			(*MetaDaten sammeln*)
			IF bStoreMetaDataInFile THEN
				FOR iMetaID :=0 TO 499 BY 1 DO
					IF arrMetaID[iMetaID]=arrDP_ID_buffer[iBuffer] THEN
						iMetaID:=500;
					ELSIF arrMetaID[iMetaID]='' THEN
						arrMetaID[iMetaID]:=arrDP_ID_buffer[iBuffer] ;
						arrMetaData[iMeta]:=arrLogDatapoints[iBuffer];
						IF arrMetaData[iMeta].sID='' THEN
							arrMetaData[iMeta].sID:=arrMetaData[iMeta].sDescription;
						END_IF
						IF arrMetaData[iMeta].sUnit='' THEN
							arrMetaData[iMeta].sUnit:='-';
						END_IF
						iMeta:=iMeta+1;
						iMetaID:=500;
			//			bStoreMeta:=TRUE;
					END_IF
				END_FOR
			END_IF
			IF iBuffer <499 THEN
				IF arrLogDatapoints[iBuffer+1].sDescription ='' AND arrLogDatapoints[iBuffer+1].sID = '' THEN
					iBuffer:=500;
				END_IF		
			END_IF				
		ELSE
			iBuffer:=500;
		END_IF
	END_FOR
ELSE
	bArrayStored:=FALSE;
END_IF

(*MetaDatenBuffern*)
IF arrMetaData[0].sDescription<>'' AND arrMetaDataBuffer[0].sDescription='' THEN
	arrMetaDataBuffer:=arrMetaData;
	iMeta:=0;
	arrMetaData:=arrMetaDataEmpty;	
END_IF

(*MetaDaten in Datei speichern*)
IF arrMetaDataBuffer[0].sDescription<>'' AND sFolderPath <>'' THEN
	CASE iState_StoreMeta OF
		0:	// Datei anlegen
			(*fbFormatMetaFilepath(
				sFormat	:= '%S\%S_%S',
				arg1	:= F_STRING(sFolderPath),
				arg2	:= F_STRING(sLMeasurement_date),
				arg3	:= F_STRING(sMetaFileName),
				sOut	=> sFilePathMeta,
				bError	=> bFormatMetaFilepath_error,
				nErrId	=> nFormatMetaFilepath_errID
			);*)
			sFilePathMeta:=CONCAT(sFolderPath,'\');
			sFilePathMeta:=CONCAT(sFilePathMeta,sLMeasurement_date);
			sFilePathMeta:=CONCAT(sFilePathMeta,sMetaFileName);
			//sFilePathMeta:=CONCAT(sFilePathMeta,'_MetaData.txt');
			fbFileOpenMeta(
				bExecute:=FALSE,
				);
			
			fbFileOpenMeta(
				sNetID:='',
				sPathName:=sFilePathMeta,
				nMode:=FOPEN_MODEAPPEND,
				//ePath:=ePath,
				bExecute:=TRUE,
				tTimeout:=T#5S,
				);
			iState_StoreMeta:=iState_StoreMeta+1;
			
		1:	// warten bis Funktionsbaustein fertig
			fbFileOpenMeta(
				bExecute:=FALSE,
				);
			IF NOT fbFileOpenMeta.bBusy THEN
				IF fbFileOpenMeta.bError THEN
					iFileOpenMeta_errID:=fbFileOpenMeta.nErrId;
					iState_StoreMeta:=0;
				ELSE
					hFileMeta:=fbFileOpenMeta.hFile;
					iFileOpenMeta_errID:=fbFileOpenMeta.nErrId;
					iState_StoreMeta:=10;
				END_IF	
			END_IF
			
		10:	// String vorbereiten
			IF arrMetaDataBuffer[iMetaBuffer].sDescription <> ''  THEN
				CASE iMetaInfo OF
					0:  sStringMeta:=CONCAT('ID=',arrMetaDataBuffer[iMetaBuffer].sID);
						sStringMeta:=CONCAT(sStringMeta,'$0A');
					1:	sStringMeta:=CONCAT('Description=',arrMetaDataBuffer[iMetaBuffer].sDescription);
						sStringMeta:=CONCAT(sStringMeta,'$0A');
					2:	sStringMeta:=CONCAT('Unit=',arrMetaDataBuffer[iMetaBuffer].sUnit);	
						sStringMeta:=CONCAT(sStringMeta,'$0A$0A');		
				END_CASE
				IF iMetaInfo>=2 THEN
					iMetaInfo:=0;
					iMetaBuffer:=iMetaBuffer+1;
				ELSE
					iMetaInfo:=iMetaInfo+1;
				END_IF	
				iState_StoreMeta:=11;
			ELSE
				iState_StoreMeta:=20;
			END_IF			
		
		11:	// Tabelle schreiben
		fbFilePutsMeta(
			sNetID:='',
			hfile:=hFileMeta,
			sLine:=sStringMeta,
			bExecute:=TRUE,
			bBusy=>bPutsMeta_busy,
			bError=>bPutsMeta_error,
			nErrId=>iPutsMeta_errorID
			);
			
		// wenn Funktionsbaustein fertig, zum nächsten Datenpunkt springen			
		IF NOT bPutsMeta_busy OR bPutsMeta_error THEN
			fbFilePutsMeta(
				bExecute:=FALSE,
				bBusy=>bPutsMeta_busy,
				bError=>bPutsMeta_error,
				nErrId=>iPutsMeta_errorID
				);
				
			IF bPutsMeta_error THEN
				nErrorMeta_LogError:=nErrorMEta_LogError+1;
			END_IF
				
			MEMSET(ADR(sStringMeta),0,255);
			iState_StoreMeta:=10;
		END_IF			
			
			
		20: // Datei schließen
			fbFileCloseMeta(
				bExecute:=FALSE,
				);
			fbFileCloseMeta(
				sNetId:='',
				hFile:=hFileMeta,
				bExecute:=TRUE,
				tTimeout:=,
				);
			iState_StoreMeta:=iState_StoreMeta+1;
			
		21: // warten bis Baustein fertig ist
			fbFileCloseMeta(
				bExecute:=FALSE,
				);
			IF NOT fbFileCloseMeta.bBusy THEN		
				IF fbFileCloseMeta.bError THEN
					iFileCloseMeta_errID:=fbFileCloseMeta.nErrId;
				END_IF
					iFileCloseMeta_errID:=fbFileCloseMeta.nErrId;
					iState_StoreMeta:=30;
			END_IF
			
		30: // Speichervorgang abgschlossen
			//bSafe_Table:=FALSE;
			iMetaBuffer:=0;
			arrMetaDataBuffer:=arrMetaDataEmpty;
			iState_StoreMeta:=0;
	END_CASE
END_IF

// Messwerte abspeichern, sofern nicht gerade die Meassdatendatei getauscht wird
IF bLogging AND hFile<>0 THEN
	bLogging_activ:=TRUE;
	CASE iStateLogging OF
	0:	// Datenpunktstring bauen
		// Dezimalunkt durch Komma ersetzen im Messwert
		IF FIND(arrDP_Value_buffer[iDatapoint_Log],'.') <>0 THEN
			arrDP_Value_buffer[iDatapoint_Log]:=REPLACE(arrDP_Value_buffer[iDatapoint_Log],',',1,FIND(arrDP_Value_buffer[iDatapoint_Log],'.')); 
		END_IF
		
		// String zusammensetzen 
			IF bLogUtcTime THEN
				// UTC
				fbFormatMeasString(
					sFormat	:= '%S%S%S%S',
					arg1	:= F_STRING(sMeasurement_date),
					arg2	:= F_STRING(sSpaces),
					arg3	:= F_STRING(sMeasurement_time),
					arg4	:= F_STRING(sDelimiter),
					sOut	=> sMeasString_temp,
					bError	=> bFormatMeasString_error,
					nErrId	=> nFormatMeasString_errID
					);
					
				IF bFormatTimestamp_error THEN
					nError_Logging:=nError_Logging+1;
				END_IF
			END_IF
			
			IF bLogLocalTime THEN
				// lokale Zeit
				fbFormatMeasString(
					sFormat	:= '%S%S%S%S%S',
					arg1	:= F_STRING(sMeasString_temp),
					arg2	:= F_STRING(sLMeasurement_date),
					arg3	:= F_STRING(sSpaces),
					arg4	:= F_STRING(sLMeasurement_time),
					arg5	:= F_STRING(sDelimiter),
					sOut	=> sMeasString_temp,
					bError	=> bFormatMeasString_error,
					nErrId	=> nFormatMeasString_errID
					);
				
				IF bFormatTimestamp_error THEN
					nError_Logging:=nError_Logging+1;
				END_IF	
			END_IF
				
			// Datenpunkte
			fbFormatMeasString(
				sFormat	:= '%S%S%S%S',
				arg1	:= F_STRING(sMeasString_temp),
				arg2	:= F_STRING(arrDP_ID_buffer[iDatapoint_Log]),
				arg3	:= F_STRING(sDelimiter),
				arg4	:= F_STRING(arrDP_Value_buffer[iDatapoint_Log]),
				sOut	=> sMeasString_temp,
				bError	=> bFormatMeasString_error,
				nErrId	=> nFormatMeasString_errID
				);

			IF bFormatTimestamp_error THEN
				nError_Logging:=nError_Logging+1;
			END_IF		
				
		// String für CSV vorbereiten
		fb_CSVbuffer(
			eCmd:=eCmd,
			putValue:=sMeasString_temp,
			pValue:=0,
			cbValue:=0,
			bCRLF:=bCRLF,
			pBuffer:=ADR(sMeasString),
			cbBuffer:=SIZEOF(sMeasString),
			cbSize=>iSize_buffer
			);
		
		sMeasString_temp:='';	
			
		// Zeilenende hinzufügen
		MEMSET(ADR(sMeasString)+iSize_buffer-2,9,1);
		sMeasString:=REPLACE(sMeasString,'$0A',2,FIND(sMeasString,'$09$0A'));
		iStateLogging:=1;
		
	1:	//Datenpunktstring schreiben
		fbFilePuts(
			sNetID:='',
			hfile:=hFile,
			sLine:=sMeasString,
			bExecute:=TRUE,
			bBusy=>bPuts_busy,
			bError=>bPuts_error,
			nErrId=>iPuts_errorID
			);
			
		bWatchdogDPwrite:=FALSE;
			
		// wenn Funktionsbaustein fertig, zum nächsten Datenpunkt springen			
		IF NOT bPuts_busy OR bPuts_error THEN
			fbFilePuts(
				bExecute:=FALSE,
				bBusy=>bPuts_busy,
				bError=>bPuts_error,
				nErrId=>iPuts_errorID
				);
				
			IF bPuts_error THEN
				nError_Logging:=nError_Logging+1;
			END_IF
				
			iDatapoint_Log:=iDatapoint_Log+1;
			MEMSET(ADR(sMeasString),0,255);
			IF arrDP_ID_buffer[iDatapoint_Log]<>'' AND iDatapoint_Log<>500 THEN
				iStateLogging:=0;
			ELSE // falls dies der letzte Datenpunkt war, Speicherzyklus beenden
				IF arrDP_ID_buffer[0]='' THEN
					iNumberOfLoggedDP:= 0;
				ELSE
					iNumberOfLoggedDP:= iDatapoint_Log;				
				END_IF
				arrDP_ID_buffer:=arrTMAXempty;
				arrDP_Value_buffer:=arrTMAXempty;
				iDatapoint_Log:=0;
				iStateLogging:=0;
				bLogging:=FALSE;
				bLogging_activ:=FALSE;
			END_IF
		END_IF
	END_CASE
END_IF

IF tLogCycleTime<T#100MS THEN
	tWatchdogDPwrite_Time:=T#500MS;
ELSE
	tWatchdogDPwrite_Time:=2*tLogCycleTime;
END_IF

fbWatchdogDPwrite(IN:=bWatchdogDPwrite, PT:= tWatchdogDPwrite_Time, Q=> , ET=> );
IF fbWatchdogDPwrite.Q THEN
	bWatchdogDPwrite:=FALSE;
	nError_Logging:=nError_Logging+1;
ELSE
	bWatchdogDPwrite:=TRUE;
END_IF

END_FUNCTION_BLOCK

// Datenlogger/FB/FB_TIME
FUNCTION_BLOCK FB_TIME
VAR
	// Allgemein
	iStateZeit					:INT;
	
	// Zeitzonenermittlung
	iState_Timezone				:INT;
	FB_GetTimeZone				:FB_GetTimeZoneInformation;
	bGetTimeZone_busy			:BOOL;
	bGetTimeZone_error			:BOOL;
	nGetTimeZone_errID			:UDINT;
	tzGetTimeZone_Info  		:ST_TimeZoneInformation;
	tzGetTimeZone_InfoTc  		:ST_TimeZoneInformation;
	nTimeZonebias				:DINT;
	
	// Erkennung der Zeitzonenänderung
	FB_TimezoneChange_Timeout	:TON;
	nTimeZoneChanging_Timeout	:UINT;
	nTimeout					:TIME:=T#1S;

	// Zeitermittlung Windows Zeit
	fbGetTime					:NT_GetTime;
	bGetTime_busy				:BOOL;
	bGetTime_error				:BOOL;
	nGetTime_errID				:UDINT;
	nGetTime_errCounter			:UDINT;
	fbTimeToUTC					:FB_TzSpecificLocalTimeToSystemTime;	
	
	// Zeitermittlung TwinCat Zeit	
	fbGetSystemTime				:GetSystemTime;
	tfTcDate					:T_Filetime;
	tTcDate						:TIMESTRUCT;
	fbUTCtoLTime				:FB_SystemTimeToTzSpecificLocalTime;
	bTimeZoneInitialized		:BOOL;
END_VAR

VAR_IN_OUT 
// ehemals Globale Variablen
	// Time	
	bUseTcTime					:BOOL;									(*Zeitbasis: fortlaufende TwinCAT-Uhr initialisiert durch Windows*)
	// Time local
	tLDate						:TIMESTRUCT;							(*aktuelles Datum lokal*)
	tfLDate						:T_Filetime;							(*aktuelles Datum lokal*)
	sLYear						:T_MaxString;							(*aktuelles Jahr lokal als String*)
	sLMonth						:T_MaxString;							(*aktueller Monat lokal als String*)
	sLDay						:T_MaxString;							(*aktueller Tag lokal als String*)
	sLHour						:T_MaxString;							(*aktuelle Stunde lokal als String*)
	sLMinute					:T_MaxString;							(*aktuelle Minute lokal als String*)
	sLSecond					:T_MaxString;							(*aktuelle Sekunde lokal als String*)
	sLMilliSecond				:T_MaxString;							(*aktulle Millisekunde lokal als String*)
	
	// Time UTC
	tDate						:TIMESTRUCT;							(*aktuelles Datum UTC*)
	tfDate						:T_Filetime;							(*aktuelles Datum UTC*)
	wDate						:LWORD;									(*aktuelles Datum UTC*)
	sYear						:T_MaxString;							(*aktuelles Jahr UTC als String*)
	sMonth						:T_MaxString;							(*aktueller Monat UTC als String*)
	sDay						:T_MaxString;							(*aktueller Tag UTC als String*)
	sHour						:T_MaxString;							(*aktuelle Stunde UTC als String*)
	sMinute						:T_MaxString;							(*aktuelle Minute UTC als String*)
	sSecond						:T_MaxString;							(*aktuelle Sekunde UTC als String*)
	sMilliSecond				:T_MaxString;							(*aktulle Millisekunde UTC als String*)
	
	// Errohandling
	nError_Time					:UINT;
END_VAR

IF NOT bUseTcTime THEN // USE Windows-Zeitbasis
	// Ermittlung der Zeitzoneninformation
		CASE iState_Timezone OF
		0:	
			FB_GetTimeZone(
				sNetID:= , 
				bExecute:=TRUE , 
				tTimeout:=T#3S , 
				bBusy=> bGetTimeZone_busy, 
				bError=> bGetTimeZone_error, 
				nErrID=> nGetTimeZone_errID, 
				tzID=> , 
				tzInfo=> );
		
			iState_Timezone:=1;
			
		1:		
			FB_GetTimeZone(
				sNetID:= , 
				bExecute:=FALSE , 
				tTimeout:=T#3S , 
				bBusy=> bGetTimeZone_busy, 
				bError=> bGetTimeZone_error, 
				nErrID=> nGetTimeZone_errID, 
				tzID=> , 
				tzInfo=> //tzGetTimeZone_Info
				);
				
			IF (bGetTimeZone_busy=FALSE) THEN
				IF NOT bGetTimeZone_error AND FB_GetTimeZone.tzInfo.standardName<>'' THEN
					tzGetTimeZone_Info:=FB_GetTimeZone.tzInfo;
					iState_Timezone:=0;
					IF tzGetTimeZone_Info.bias<>nTimeZonebias THEN
						nTimeZonebias:=tzGetTimeZone_Info.bias;
						iStateZeit:=3;
					END_IF
				ELSE
					nError_Time:=nError_Time+1;
					iState_Timezone:=0;
				END_IF
			END_IF
		END_CASE
	
	
		CASE iStateZeit OF
		0:
			(*Zeit auslesen*)
			fbGetTime(
				NETID		:= '',
				START		:= TRUE,
				TMOUT		:= T#2s,
				BUSY		=>bGetTime_busy ,
				ERR			=>bGetTime_error ,
				ERRID		=>nGetTime_errID ,
				TIMESTR		=>
			);
			
			fbGetTime(
				START		:= FALSE,
			);
			fbGetTime(
				START		:= TRUE,
			);
			iStateZeit:=1;
			
		1:
			fbGetTime(
				START		:= FALSE,
				BUSY		=>bGetTime_busy ,
				ERR			=>bGetTime_error ,
				ERRID		=>nGetTime_errID ,
			);
			
			IF NOT fbGetTime.BUSY AND NOT fbGetTime.ERR  THEN
				(*aktuelles Datum lokal*)
				tLDate	:= fbGetTime.TIMESTR;
				tfLDate	:= SYSTEMTIME_TO_FILETIME(tLDATE);
				
				(* lokale Zeit in String übersetzen*)
				sLYear			:= DWORD_TO_DECSTR(tLDate.wYear, 4);
				sLMonth			:= DWORD_TO_DECSTR(tLDate.wMonth, 2);
				sLDay			:= DWORD_TO_DECSTR(tLDate.wDay, 2);
				sLHour			:= DWORD_TO_DECSTR(tLDate.wHour, 2);
				sLMinute		:= DWORD_TO_DECSTR(tLDate.wMinute, 2);
				sLSecond		:= DWORD_TO_DECSTR(tLDate.wSecond, 2);
				sLMilliSecond	:= DWORD_TO_DECSTR(tLDate.wMilliseconds, 3);
				
				(*aktuelles Datum UTC*)
				fbTimeToUTC(
					in:= tlDate, 
					tzInfo:= tzGetTimeZone_Info, 
					out=> tDate, 
					eTzID=> , 
					bB=> );
				tfDate	:=	SYSTEMTIME_TO_FILETIME(tDate);
				MEMCPY(ADR(wDate)+4,ADR(tfDate.dwHighDateTime),4);
				MEMCPY(ADR(wDate),ADR(tfDate.dwLowDateTime),4);		
				
				(*UTC Zeit in String übersetzen*)
				sYear			:= DWORD_TO_DECSTR(tDate.wYear, 4);
				sMonth			:= DWORD_TO_DECSTR(tDate.wMonth, 2);
				sDay			:= DWORD_TO_DECSTR(tDate.wDay, 2);
				sHour			:= DWORD_TO_DECSTR(tDate.wHour, 2);
				sMinute			:= DWORD_TO_DECSTR(tDate.wMinute, 2);
				sSecond			:= DWORD_TO_DECSTR(tDate.wSecond, 2);
				sMilliSecond	:= DWORD_TO_DECSTR(tDate.wMilliseconds, 3);
				
				iStateZeit:=0;	
			ELSIF NOT fbGetTime.BUSY AND fbGetTime.ERR  THEN
				iStateZeit:=0;
				nError_Time:=nError_Time+1;
				nGetTime_errCounter:=nGetTime_errCounter+1;		
			END_IF
		
		3:	// Timeout bei Zeitzonenänderung
			FB_TimezoneChange_Timeout(IN:= TRUE, PT:= nTimeout , Q=> , ET=> );
			IF FB_TimezoneChange_Timeout.Q THEN
				iStateZeit:=0;
				FB_TimezoneChange_Timeout(IN:= FALSE, PT:= nTimeout , Q=> , ET=> );
				fbGetTime(
					START		:= FALSE,
				);	
			END_IF
		END_CASE		
ELSE	// USE TwinCat Zeitbasis
	CASE iState_Timezone OF
	// Ermittlung der Zeitzoneninformation
	0:	
		FB_GetTimeZone(
			sNetID:= , 
			bExecute:=TRUE , 
			tTimeout:=T#3S , 
			bBusy=> bGetTimeZone_busy, 
			bError=> bGetTimeZone_error, 
			nErrID=> nGetTimeZone_errID, 
			tzID=> , 
			tzInfo=> );
	
		iState_Timezone:=1;
		
	1:		
		FB_GetTimeZone(
			sNetID:= , 
			bExecute:=FALSE , 
			tTimeout:=T#3S , 
			bBusy=> bGetTimeZone_busy, 
			bError=> bGetTimeZone_error, 
			nErrID=> nGetTimeZone_errID, 
			tzID=> , 
			tzInfo=> tzGetTimeZone_Info
			);
			
		IF (bGetTimeZone_busy=FALSE) THEN
			IF NOT bGetTimeZone_error THEN
				tzGetTimeZone_InfoTc:=FB_GetTimeZone.tzInfo;
				iState_Timezone:=0;
			ELSE
				nError_Time:=nError_Time+1;
				iState_Timezone:=0;
			END_IF
			bTimeZoneInitialized :=TRUE;
		END_IF	
	END_CASE	
	
	IF bTimeZoneInitialized THEN
	// Errechnung der UTC auf Basis der TwinCat Zeit
		(*aktuelles Datum UTC TwinCat*)
		fbGetSystemTime(timeLoDW=>tfTcDate.dwLowDateTime , timeHiDW=> tfTcDate.dwHighDateTime);
		tTcDate	:=	FILETIME_TO_SYSTEMTIME(tfTcDate);
		
		(*aktuelles Datum lokal*)
		fbUTCtoLTime(
			in:= tTcDate, 
			tzInfo:= tzGetTimeZone_InfoTc, 
			out=> tLDate, 
			eTzID=> , 
			bB=> );		
		tfLDate	:= SYSTEMTIME_TO_FILETIME(tLDATE);
		
		(* lokale Zeit in String übersetzen*)
		sLYear			:= DWORD_TO_DECSTR(tLDate.wYear, 4);
		sLMonth			:= DWORD_TO_DECSTR(tLDate.wMonth, 2);
		sLDay			:= DWORD_TO_DECSTR(tLDate.wDay, 2);
		sLHour			:= DWORD_TO_DECSTR(tLDate.wHour, 2);
		sLMinute		:= DWORD_TO_DECSTR(tLDate.wMinute, 2);
		sLSecond		:= DWORD_TO_DECSTR(tLDate.wSecond, 2);
		sLMilliSecond	:= DWORD_TO_DECSTR(tLDate.wMilliseconds, 3);
		
		(*aktuelles Datum UTC*)	
		tfDate:=tfTcDate;	
		tDate	:=	FILETIME_TO_SYSTEMTIME(tfDate);
		MEMCPY(ADR(wDate)+4,ADR(tfDate.dwHighDateTime),4);
		MEMCPY(ADR(wDate),ADR(tfDate.dwLowDateTime),4);		
		
		(*UTC Zeit in String übersetzen*)
		sYear			:= DWORD_TO_DECSTR(tDate.wYear, 4);
		sMonth			:= DWORD_TO_DECSTR(tDate.wMonth, 2);
		sDay			:= DWORD_TO_DECSTR(tDate.wDay, 2);
		sHour			:= DWORD_TO_DECSTR(tDate.wHour, 2);
		sMinute			:= DWORD_TO_DECSTR(tDate.wMinute, 2);
		sSecond			:= DWORD_TO_DECSTR(tDate.wSecond, 2);
		sMilliSecond	:= DWORD_TO_DECSTR(tDate.wMilliseconds, 3);
	END_IF	
END_IF

END_FUNCTION_BLOCK

// Datenlogger/FB_Datenlogger
FUNCTION_BLOCK FB_Datenlogger
VAR_INPUT
	arrLogDatapoints			:ARRAY [0..499] OF Log_Datapoint;		(*Logging Input*)
//	arrDatenpunkt_ID			:ARRAY [0..99] OF T_MaxString;			(*Beschreibung der Datenpunkte*)
//	arrDatenpunkt				:ARRAY [0..99] OF T_MaxString;			(*Messwerte der Datenpunkte*)
	sPathName				 	:T_MaxString:='C:\Messdaten\'; 			(*Pfad der Messdaten festlegen (default: C:\Messdaten\, nur der letzte Unterordner wird (falls nicht vorhanden) erstellt*)
	tZykluszeit					:TIME:=T#10S;							(*Messzykluszeit (default: 10s), 0 entspricht so schnell wie möglich*)
	bExecute					:BOOL:=TRUE;							(*externe (De)aktivierung der Loggingfunktion (default: aktiviert)*)
	bUseTwinCatTimeBase			:BOOL:=FALSE;							(*Zeit auf Basis der fortlaufenden TwinCAT-Uhr intialisiert durch Windows (default: deaktiviert); zu verwenden wenn die WindowsZeit nicht netzwerkseitig synchronisiert wird*)
	bLocalTimeLogging			:BOOL:=TRUE;							(*lokale Zeit mitloggen (default: aktiviert)*)
	bOldOutputFile				:BOOL:=FALSE;							(*FALSE(default)OutputFile:"idTABvalue"; TRUE(oldFormat):OutputFile: "DescriptionTAB[unit]TABvalue --> no Meta"*)
END_VAR
VAR_OUTPUT
	bArrayStored				:BOOL;									(*Flag, Loggarray in Puffer übertragen*)
	sLogFilePath				:STRING;								(*Path of actual LogFile*)
	arrLoggedDatapoints			:ARRAY [0..499] OF Log_Datapoint;		(*Array of Logged Datapoints*)
	iNumberOfLoggedDatapoints	:INT;									(*information of Loged Datapoints*)
	nErrorCounter				:UINT;									(*Anzahl aufgelaufener Fehler*)
END_VAR
VAR
	FB_TIME						:FB_TIME;								(*Funktionsbaustein für die Zeitsteuerung*)
	FB_FOLDER					:FB_FOLDER;								(*Funktionsbaustein für die Ordnererstellung*)
	FB_FILE						:FB_FILE;								(*Funktionsbaustein für die Dateierstellung*)
	FB_LOGGING					:FB_LOGGING;							(*Funktionsbaustein für das Schreiben der Messdaten*)
END_VAR
VAR
	bUtcTimeLogging				:BOOL:=TRUE;							(*UTC mitloggen (default: aktiviert)*)
// ehemals Globale Variablen
// General	
	arrDatapoint_ID				:ARRAY [0..499] OF T_MaxString;			(*Beschreibung der Datenpunkte*)
	arrDatapoint_Value			:ARRAY [0..499] OF T_MaxString;			(*Messwerte der Datenpunkte*)
	sDataPath					:T_MaxString:='C:\Messdaten\'; 			(*Pfad der Messdaten*)
	tLogCycleTime				:TIME:=T#10S;							(*Messzyklusvorgabe*)

// Time	
	bUseTcTime					:BOOL;									(*Zeitbasis: fortlaufende TwinCAT-Uhr initialisiert durch Windows*)
	// Time local
	tLDate						:TIMESTRUCT;							(*aktuelles Datum lokal*)
	tfLDate						:T_Filetime;							(*aktuelles Datum lokal*)
	sLYear						:T_MaxString;							(*aktuelles Jahr lokal als String*)
	sLMonth						:T_MaxString;							(*aktueller Monat lokal als String*)
	sLDay						:T_MaxString;							(*aktueller Tag lokal als String*)
	sLHour						:T_MaxString;							(*aktuelle Stunde lokal als String*)
	sLMinute					:T_MaxString;							(*aktuelle Minute lokal als String*)
	sLSecond					:T_MaxString;							(*aktuelle Sekunde lokal als String*)
	sLMilliSecond				:T_MaxString;							(*aktulle Millisekunde lokal als String*)
	
	// Time UTC
	tDate						:TIMESTRUCT;							(*aktuelles Datum UTC*)
	tfDate						:T_Filetime;							(*aktuelles Datum UTC*)
	wDate						:LWORD;									(*aktuelles Datum UTC*)
	sYear						:T_MaxString;							(*aktuelles Jahr UTC als String*)
	sMonth						:T_MaxString;							(*aktueller Monat UTC als String*)
	sDay						:T_MaxString;							(*aktueller Tag UTC als String*)
	sHour						:T_MaxString;							(*aktuelle Stunde UTC als String*)
	sMinute						:T_MaxString;							(*aktuelle Minute UTC als String*)
	sSecond						:T_MaxString;							(*aktuelle Sekunde UTC als String*)
	sMilliSecond				:T_MaxString;							(*aktulle Millisekunde UTC als String*)
	
	
// File and Folder
	// allgemein
	iStateFolder				:INT;									(*Case Auswahl der Ordnererzeugung*)
	arrLastFolder				:ARRAY [0..2] OF STRING;				(*letzter erzeugter Datumsordner*)
	sFolderPath					:T_MaxString;							(*Pfad, zum Messdatenordner*)
	sFilePath					:T_MaxString;							(*Pfad zur Messdatendatei*)
	
	// Statusvariablen der Dateierstellung
	sLastFile_Changed			:T_MaxString:='99';						(*Minute der letzten Änderung des verwedndeten Datenfiles*)
	sLastFile_Opened			:T_MaxString:='99';						(*Minute des letzten geöffneten Datenfiles*)

	// Dateireferenzen	
	hFile						:UINT;									(*Referenz der aktuellen Messdatendatei*)
	hFile_Close					:UINT;									(*Referenz der zu schließenden Messdatendatei*)
	arrhFile_Open				:ARRAY [0..10] OF UINT;					(*Referenz-Array der geöffneten Messdatendatein*)		

// Logging
	wNextMeasurement			:LWORD;									(*Zeit des nächsten vorgesehenen Loggings*)
	bLogging_activ				:BOOL;									(*Flag; zeigt an, ob gerade Werte geschrieben werden*)
	bLogUtcTime					:BOOL;									(*UTC Zeit mitloggen*)
	bLogLocalTime				:BOOL;									(*lokale Zeit mitloggen*)
	
// Errohandling
	nError_Time					:UINT;
	nError_Folder				:UINT;
	nError_File_Open			:UINT;
	nError_File_Close			:UINT;	
	nError_File_Change			:UINT;		
	nError_Logging				:UINT;	
	nError_Datalogger			:UINT;
END_VAR

// Verknüpfung der Eingänge auf die globalen Variablen
// zur Nutzung des Funktionsbausteins aus in bestehenden Projekten
//arrDatapoint_ID			:=arrDatenpunkt_ID;
//arrDatapoint_Value		:=arrDatenpunkt;
sDataPath				:=sPathName;
tLogCycleTime			:=tZykluszeit;
bLogUtcTime				:=bUtcTimeLogging;			
bLogLocalTime			:=bLocalTimeLogging;
bUseTcTime				:=bUseTwinCatTimeBase;		

FB_TIME(
	bUseTcTime:= bUseTcTime, 
	tLDate:= tLDate, 
	tfLDate:= tfLDate, 
	sLYear:= sLYear, 
	sLMonth:= sLMonth, 
	sLDay:= sLDay, 
	sLHour:= sLHour, 
	sLMinute:= sLMinute, 
	sLSecond:= sLSecond, 
	sLMilliSecond:= sLMilliSecond, 
	tDate:= tDate, 
	tfDate:= tfDate, 
	wDate:= wDate, 
	sYear:= sYear, 
	sMonth:= sMonth, 
	sDay:= sDay, 
	sHour:= sHour, 
	sMinute:= sMinute, 
	sSecond:= sSecond, 
	sMilliSecond:= sMilliSecond, 
	nError_Time:= nError_Time);
	
IF NOT bExecute  THEN // Rücksetzen des Loggers in Ausgangsstellung
	IF bLogging_activ THEN
		FB_LOGGING(
			arrLogDatapoints:=arrLogDatapoints,
			bArrayStored:=bArrayStored,
//			arrDatapoint_ID:= arrDatapoint_ID, 
//			arrDatapoint_Value:= arrDatapoint_Value, 
			tLogCycleTime:= tLogCycleTime, 
			sLYear:= sLYear, 
			sLMonth:= sLMonth, 
			sLDay:= sLDay, 
			sLHour:= sLHour, 
			sLMinute:= sLMinute, 
			sLSecond:= sLSecond, 
			sLMilliSecond:= sLMilliSecond, 
			wDate:= wDate, 
			sYear:= sYear, 
			sMonth:= sMonth, 
			sDay:= sDay, 
			sHour:= sHour, 
			sMinute:= sMinute, 
			sSecond:= sSecond, 
			sMilliSecond:= sMilliSecond, 
			sFolderPath:=sFolderPath,
			hFile:= hFile, 
			wNextMeasurement:= wNextMeasurement, 
			bLogging_activ:= bLogging_activ, 
			bLogUtcTime:= bLogUtcTime, 
			bLogLocalTime:= bLogLocalTime,
			bOldOutputFile :=bOldOutputFile,
			nError_Logging:= nError_Logging, 
			nError_Datalogger:= nError_Datalogger,
			iNumberOfLoggedDP=>iNumberOfLoggedDatapoints,
			arrLoggedDatapoints=>arrLoggedDatapoints);
			
	ELSIF hFile <> 0 THEN
		// Datei freigeben	
		sLastFile_Changed			:='97';
		sLastFile_Opened			:='97';
		hFile_Close					:=hFile;
		FB_FILE(
			tfDate:= tfDate, 
			sYear:= sYear, 
			sMonth:= sMonth, 
			sDay:= sDay, 
			sHour:= sHour, 
			sMinute:= sMinute, 
			sSecond:= sSecond, 
			sMilliSecond:= sMilliSecond, 
			sFolderPath:= sFolderPath, 
			sFilePath:= sFilePath, 
			sLastFile_Changed:= sLastFile_Changed, 
			sLastFile_Opened:= sLastFile_Opened, 
			hFile:= hFile, 
			hFile_Close:= hFile_Close, 
			arrhFile_Open:= arrhFile_Open, 
			bLogging_activ:= bLogging_activ, 
			nError_File_Open:= nError_File_Open, 
			nError_File_Close:= nError_File_Close, 
			nError_File_Change:= nError_File_Change);
		
		// Werte für Loggerneustart Rücksetzen
		wNextMeasurement			:=0;
		iStateFolder				:=0;
		arrLastFolder[0]			:='0';
		arrLastFolder[1]			:='0';
		arrLastFolder[2]			:='0';
		sFolderPath					:='';
		sFilePath					:='';
		bArrayStored:=TRUE;
	ELSE
		bArrayStored:=FALSE;	
	END_IF

ELSE	// Aufruf der Funktionsbausteine
	FB_FOLDER(
		sDataPath:= sDataPath, 
		tfDate:= tfDate, 
		wDate:= wDate, 
		sYear:= sYear, 
		iStateFolder:= iStateFolder, 
		arrLastFolder:= arrLastFolder, 
		sFolderPath:= sFolderPath, 
		nError_Folder:= nError_Folder);
	FB_FILE(
		tfDate:= tfDate, 
		sYear:= sYear, 
		sMonth:= sMonth, 
		sDay:= sDay, 
		sHour:= sHour, 
		sMinute:= sMinute, 
		sSecond:= sSecond, 
		sMilliSecond:= sMilliSecond, 
		sFolderPath:= sFolderPath, 
		sFilePath:= sFilePath, 
		sLastFile_Changed:= sLastFile_Changed, 
		sLastFile_Opened:= sLastFile_Opened, 
		hFile:= hFile, 
		hFile_Close:= hFile_Close, 
		arrhFile_Open:= arrhFile_Open, 
		bLogging_activ:= bLogging_activ, 
		nError_File_Open:= nError_File_Open, 
		nError_File_Close:= nError_File_Close, 
		nError_File_Change:= nError_File_Change);
		
	FB_LOGGING(
		arrLogDatapoints:=arrLogDatapoints,
		bArrayStored:=bArrayStored,
//		arrDatapoint_ID:= arrDatapoint_ID, 
//		arrDatapoint_Value:= arrDatapoint_Value, 
		tLogCycleTime:= tLogCycleTime, 
		sLYear:= sLYear, 
		sLMonth:= sLMonth, 
		sLDay:= sLDay, 
		sLHour:= sLHour, 
		sLMinute:= sLMinute, 
		sLSecond:= sLSecond, 
		sLMilliSecond:= sLMilliSecond, 
		wDate:= wDate, 
		sYear:= sYear, 
		sMonth:= sMonth, 
		sDay:= sDay, 
		sHour:= sHour, 
		sMinute:= sMinute, 
		sSecond:= sSecond, 
		sMilliSecond:= sMilliSecond, 
		sFolderPath:=sFolderPath,
		hFile:= hFile, 
		wNextMeasurement:= wNextMeasurement, 
		bLogging_activ:= bLogging_activ, 
		bLogUtcTime:= bLogUtcTime, 
		bLogLocalTime:= bLogLocalTime, 
		bOldOutputFile:=bOldOutputFile,
		nError_Logging:= nError_Logging, 
		nError_Datalogger:= nError_Datalogger,
		iNumberOfLoggedDP=>iNumberOfLoggedDatapoints,
		arrLoggedDatapoints=>arrLoggedDatapoints);		
END_IF

IF sFilePath <> '' THEN
	sLogFilePath:=sFilePath;
END_IF
nError_Datalogger:=nError_Time+nError_Folder+nError_File_Open+nError_File_Change+nError_File_Close+nError_Logging;
nErrorCounter	:=nError_Datalogger;

END_FUNCTION_BLOCK

// Functions/FUN_ByteArrToString
FUNCTION FUN_ByteArrToString :STRING
VAR_INPUT
	arrTempBytes:ARRAY [0..7] OF BYTE;
	iDatatyp 	:Datatyp;
	bHex		:BOOL;
END_VAR
VAR
	sTempBYTE :BYTE;
	sTempWORD :WORD;
	sTempDWORD :DWORD;
	sTempSINT :SINT;
	sTempINT :INT;
	sTempDINT :DINT;
	sTempLINT :LINT;
	sTempUSINT :USINT;
	sTempUINT :UINT;
	sTempUDINT :UDINT;
	sTempULINT :ULINT;
	sTempREAL :REAL;
	sTempLREAL :LREAL;
	sTempBOOL :BYTE;
	sTempEnum :BYTE;
END_VAR

CASE iDatatyp OF
0: // NO_DATA_TYP_DEFINED

1:	// BYTE
	MEMCPY(ADR(sTempBYTE),ADR(arrTempBytes),SIZEOF(sTempBYTE));
	IF bHex THEN
		FUN_ByteArrToString := BYTE_TO_HEXSTR(sTempBYTE,0,FALSE);
	ELSE
		FUN_ByteArrToString := BYTE_TO_STRING(sTempBYTE);
	END_IF
		
	
2: // WORD
	MEMCPY(ADR(sTempWORD), ADR(arrTempBytes), SIZEOF(sTempWORD));	
	IF bHex THEN
		FUN_ByteArrToString := WORD_TO_HEXSTR(sTempWORD,0,FALSE);
	ELSE
		FUN_ByteArrToSTring := WORD_TO_STRING(sTempWORD);
	END_IF
	
3: // DWORD
	MEMCPY(ADR(sTempDWORD), ADR(arrTempBytes), SIZEOF(sTempDWORD));	
	IF bHex THEN
		FUN_ByteArrToString := DWORD_TO_HEXSTR(sTempDWORD,0,FALSE);
	ELSE
		FUN_ByteArrToSTring := DWORD_TO_STRING(sTempDWORD);
	END_IF

4: // SINT
	MEMCPY(ADR(sTempSINT), ADR(arrTempBytes), SIZEOF(sTempSINT));	
	IF bHex THEN
		FUN_ByteArrToSTring := DATA_TO_HEXSTR(pData := ADR(sTempSINT), cbData:=SIZEOF(sTempSINT),bLoCase:=FALSE);
	ELSE
		FUN_ByteArrToSTring := SINT_TO_STRING(sTempSINT);		
	END_IF
		
5: // INT
	MEMCPY(ADR(sTempINT), ADR(arrTempBytes), SIZEOF(sTempINT));	
	IF bHex THEN
		FUN_ByteArrToSTring := DATA_TO_HEXSTR(pData := ADR(sTempINT), cbData:=SIZEOF(sTempINT),bLoCase:=FALSE);
	ELSE
		FUN_ByteArrToSTring := INT_TO_STRING(sTempINT);		
	END_IF
	
6: // DINT
	MEMCPY(ADR(sTempDINT), ADR(arrTempBytes), SIZEOF(sTempDINT));	
	IF bHex THEN
		FUN_ByteArrToSTring := DATA_TO_HEXSTR(pData := ADR(sTempDINT), cbData:=SIZEOF(sTempDINT),bLoCase:=FALSE);
	ELSE
		FUN_ByteArrToSTring := DINT_TO_STRING(sTempDINT);		
	END_IF
	
7: // LINT
	MEMCPY(ADR(sTempLINT), ADR(arrTempBytes), SIZEOF(sTempLINT));	
	IF bHex THEN
		FUN_ByteArrToSTring := DATA_TO_HEXSTR(pData := ADR(sTempLINT), cbData:=SIZEOF(sTempLINT),bLoCase:=FALSE);
	ELSE
		FUN_ByteArrToSTring := LINT_TO_STRING(sTempLINT);
	END_IF
	
8: // USINT
	MEMCPY(ADR(sTempUSINT), ADR(arrTempBytes), SIZEOF(sTempUSINT));	
	IF bHex THEN
		FUN_ByteArrToSTring := DATA_TO_HEXSTR(pData := ADR(sTempUSINT), cbData:=SIZEOF(sTempUSINT),bLoCase:=FALSE);
	ELSE
		FUN_ByteArrToSTring := USINT_TO_STRING(sTempUSINT);		
	END_IF
	
9: // UINT
	MEMCPY(ADR(sTempUINT), ADR(arrTempBytes), SIZEOF(sTempUINT));	
	IF bHex THEN
		FUN_ByteArrToSTring := DATA_TO_HEXSTR(pData := ADR(sTempUINT), cbData:=SIZEOF(sTempUINT),bLoCase:=FALSE);
	ELSE
		FUN_ByteArrToSTring := UINT_TO_STRING(sTempUINT);		
	END_IF
	
10: // UDINT
	MEMCPY(ADR(sTempUDINT), ADR(arrTempBytes), SIZEOF(sTempUDINT));	
	IF bHex THEN
		FUN_ByteArrToSTring := DATA_TO_HEXSTR(pData := ADR(sTempUDINT), cbData:=SIZEOF(sTempUDINT),bLoCase:=FALSE);
	ELSE
		FUN_ByteArrToSTring := UDINT_TO_STRING(sTempUDINT);
	END_IF
	
11: // ULINT
	MEMCPY(ADR(sTempULINT), ADR(arrTempBytes), SIZEOF(sTempULINT));	
	IF bHex THEN
		FUN_ByteArrToSTring := DATA_TO_HEXSTR(pData := ADR(sTempULINT), cbData:=SIZEOF(sTempULINT),bLoCase:=FALSE);
	ELSE
		FUN_ByteArrToSTring := ULINT_TO_STRING(sTempULINT);		
	END_IF
	
12: // REAL
	MEMCPY(ADR(sTempREAL), ADR(arrTempBytes), SIZEOF(sTempREAL));	
	IF bHex THEN
		FUN_ByteArrToSTring := DATA_TO_HEXSTR(pData := ADR(sTempREAL), cbData:=SIZEOF(sTempREAL),bLoCase:=FALSE);
	ELSE
		FUN_ByteArrToSTring := REAL_TO_STRING(sTempREAL);		
	END_IF
	
13: // LREAL
	MEMCPY(ADR(sTempLREAL), ADR(arrTempBytes), SIZEOF(sTempLREAL));	
	IF bHex THEN
		FUN_ByteArrToSTring := DATA_TO_HEXSTR(pData := ADR(sTempLREAL), cbData:=SIZEOF(sTempLREAL),bLoCase:=FALSE);
	ELSE
		FUN_ByteArrToSTring := LREAL_TO_STRING(sTempLREAL);		
	END_IF
	
14: // BOOL->Byte
	MEMCPY(ADR(sTempBOOL), ADR(arrTempBytes), SIZEOF(sTempBOOL));	
	IF bHex THEN
		FUN_ByteArrToSTring := DATA_TO_HEXSTR(pData := ADR(sTempBOOL), cbData:=SIZEOF(sTempBOOL),bLoCase:=FALSE);
	ELSE
		FUN_ByteArrToSTring := BYTE_TO_STRING(sTempBOOL);		
	END_IF
	
15: // ENUM->Byte
	MEMCPY(ADR(sTempENUM), ADR(arrTempBytes), SIZEOF(sTempENUM));	
	IF bHex THEN
		FUN_ByteArrToSTring := DATA_TO_HEXSTR(pData := ADR(sTempENUM), cbData:=SIZEOF(sTempENUM),bLoCase:=FALSE);
	ELSE
		FUN_ByteArrToSTring := BYTE_TO_STRING(sTempENUM);	
	END_IF
	
END_CASE

END_FUNCTION

// Functions/FUN_DatatypSize
FUNCTION FUN_DatatypSize : UINT
VAR_INPUT
	iDatatyp :Datatyp;
END_VAR
VAR
END_VAR

CASE iDatatyp OF
0: // NOT DEFINED
	FUN_DatatypSize:=0;	
1: // BYTE
	FUN_DatatypSize:=1;
2: // WORD
	FUN_DatatypSize:=2;
3: // DWORD
	FUN_DatatypSize:=4;
4: // SINT
	FUN_DatatypSize:=1;
5: // INT
	FUN_DatatypSize:=2;
6: // DINT
	FUN_DatatypSize:=4;
7: // LINT
	FUN_DatatypSize:=8;
8: // USINT
	FUN_DatatypSize:=1;
9: // UINT
	FUN_DatatypSize:=2;
10: // UDINT
	FUN_DatatypSize:=4;
11: // ULINT
	FUN_DatatypSize:=8;
12: // REAL
	FUN_DatatypSize:=4;
13: // LREAL
	FUN_DatatypSize:=8;
14: // BOOL->Byte
	FUN_DatatypSize:=1;
15: // ENUM->Byte
	FUN_DatatypSize:=1;
END_CASE

END_FUNCTION

// Functions/FUN_StringToByteArr
FUNCTION FUN_StringToByteArr : ARRAY [0..7] OF BYTE
VAR_INPUT
	sTempValue	:STRING;
	iDatatyp 	:Datatyp;
END_VAR
VAR
	sTempBYTE :BYTE;
	sTempWORD :WORD;
	sTempDWORD :DWORD;
	sTempSINT :SINT;
	sTempINT :INT;
	sTempDINT :DINT;
	sTempLINT :LINT;
	sTempUSINT :USINT;
	sTempUINT :UINT;
	sTempUDINT :UDINT;
	sTempULINT :ULINT;
	sTempREAL :REAL;
	sTempLREAL :LREAL;
	sTempBOOL :BYTE;
	sTempEnum :BYTE;
END_VAR

CASE iDatatyp OF
0: // NO_DATA_TYP_DEFINED

1:	// BYTE
	sTempBYTE := STRING_TO_BYTE(sTempValue);
	MEMCPY(ADR(FUN_StringToByteArr),ADR(sTempBYTE),SIZEOF(sTempBYTE));
2: // WORD
	sTempWORD := STRING_TO_WORD(sTempValue);
	MEMCPY(ADR(FUN_StringToByteArr),ADR(sTempWORD),SIZEOF(sTempWORD));
3: // DWORD
	sTempDWORD := STRING_TO_DWORD(sTempValue);
	MEMCPY(ADR(FUN_StringToByteArr),ADR(sTempDWORD),SIZEOF(sTempDWORD));
4: // SINT
	sTempSINT := STRING_TO_SINT(sTempValue);
	MEMCPY(ADR(FUN_StringToByteArr),ADR(sTempSINT),SIZEOF(sTempSINT));
5: // INT
	sTempINT := STRING_TO_INT(sTempValue);
	MEMCPY(ADR(FUN_StringToByteArr),ADR(sTempINT),SIZEOF(sTempINT));
6: // DINT
	sTempDINT := STRING_TO_DINT(sTempValue);
	MEMCPY(ADR(FUN_StringToByteArr),ADR(sTempDINT),SIZEOF(sTempDINT));
7: // LINT
	sTempLINT := STRING_TO_LINT(sTempValue);
	MEMCPY(ADR(FUN_StringToByteArr),ADR(sTempLINT),SIZEOF(sTempLINT));
8: // USINT
	sTempUSINT := STRING_TO_USINT(sTempValue);
	MEMCPY(ADR(FUN_StringToByteArr),ADR(sTempUSINT),SIZEOF(sTempUSINT));
9: // UINT
	sTempUINT := STRING_TO_UINT(sTempValue);
	MEMCPY(ADR(FUN_StringToByteArr),ADR(sTempUINT),SIZEOF(sTempUINT));
10: // UDINT
	sTempUDINT := STRING_TO_UDINT(sTempValue);
	MEMCPY(ADR(FUN_StringToByteArr),ADR(sTempUDINT),SIZEOF(sTempUDINT));
11: // ULINT
	sTempULINT := STRING_TO_ULINT(sTempValue);
	MEMCPY(ADR(FUN_StringToByteArr),ADR(sTempULINT),SIZEOF(sTempULINT));
12: // REAL
	sTempREAL := STRING_TO_REAL(sTempValue);
	MEMCPY(ADR(FUN_StringToByteArr),ADR(sTempREAL),SIZEOF(sTempREAL));
13: // LREAL
	sTempLREAL := STRING_TO_LREAL(sTempValue);
	MEMCPY(ADR(FUN_StringToByteArr),ADR(sTempLREAL),SIZEOF(sTempLREAL));
14: // BOOL->Byte
	sTempBOOL := STRING_TO_BYTE(sTempValue);
	MEMCPY(ADR(FUN_StringToByteArr),ADR(sTempBOOL),SIZEOF(sTempBOOL));
15: // ENUM->Byte
	sTempEnum := STRING_TO_BYTE(sTempValue);
	MEMCPY(ADR(FUN_StringToByteArr),ADR(sTempEnum),SIZEOF(sTempEnum));	
END_CASE

END_FUNCTION

// Timetable/FB_TimeTable
FUNCTION_BLOCK FB_TimeTable
VAR_INPUT
//	nInputValue					:LREAL;		
	arrTimeControl				:ARRAY [0..49] OF Struct_TimeTable;
END_VAR

VAR_OUTPUT
	nOutputValue				:LREAL;
	bValueChanged				:BOOL;
END_VAR
VAR
	wLastMinute					:WORD;
	iRow						:INT;
	
	// Zeitermittlung Windows Zeit
	iStateZeit					:INT;
	fbGetTime					:NT_GetTime;
	bGetTime_busy				:BOOL;
	bGetTime_error				:BOOL;
	nGetTime_errID				:UDINT;
	
	// Time local
	tLDate						:TIMESTRUCT;				(*aktuelles Datum lokal*)
	

	// Tabelle abspeichern
	arrTimeControlSafed			:ARRAY [0..49] OF Struct_TimeTable;
	bSafe_Table					:BOOL;
	iState_safe					:INT;
	sFilePath					:T_MaxString:='C:\Timetable.txt';
	// Datei öffnen
	bOpenFile					:BOOL;
	fbFileOpen					:FB_FileOpen;
	iFileOpen_errID				:UDINT;
	hFile						:UINT;
	// Datei schließen
	bCloseFile					:BOOL;
	fbFileClose					:FB_FileClose;
	iFileClose_errID			:UDINT;
	// Daten schreiben
	iRow_safe					:INT;
	sString						:T_MaxString;
	fbFilePuts       			:FB_FilePuts;
	bPuts_busy					:BOOL;
	bPuts_error					:BOOL;
	iPuts_errorID				:UDINT;
	nError_LogError				:INT;
	
	// String bauen
	fbFormatString				:FB_FormatString;
	bFormatString_error			:BOOL;
	nFormatString_errID			:UDINT;
	sDelimiter					:T_MaxString:='$09';		(*$09 = Tab stop*)
	sSpaces						:T_MaxString:='$20';		(*$20 = Leerzeichen*)

	// Datenpunktstring für schreiben vorbereiten
	fb_CSVbuffer				:FB_CSVMemBufferWriter;
	eCmd    					:E_EnumCmdType := eEnumCmd_First;
	putValue 					:T_MaxString ;
	pValue  					:POINTER TO BYTE := 0;
	cbValue  					:UDINT := 0;
	bCRLF   					:BOOL :=TRUE;
	pBuffer  					:POINTER TO BYTE;
	cbBuffer 					:UDINT;
	iSize_buffer				:UDINT;	
END_VAR

// Zeit ermitteln
	CASE iStateZeit OF
	0:
		(*Zeit auslesen*)
		fbGetTime(
			NETID		:= '',
			START		:= TRUE,
			TMOUT		:= T#2s,
			BUSY		=>bGetTime_busy ,
			ERR			=>bGetTime_error ,
			ERRID		=>nGetTime_errID ,
			TIMESTR		=>
		);
		
		fbGetTime(
			START		:= FALSE,
		);
		fbGetTime(
			START		:= TRUE,
		);
		iStateZeit:=1;
		
	1:
		fbGetTime(
			START		:= FALSE,
			BUSY		=>bGetTime_busy ,
			ERR			=>bGetTime_error ,
			ERRID		=>nGetTime_errID ,
		);
		
		IF NOT fbGetTime.BUSY AND NOT fbGetTime.ERR  THEN
			(*aktuelles Datum lokal*)
			tLDate	:= fbGetTime.TIMESTR;
			iStateZeit:=0;	
		ELSIF NOT fbGetTime.BUSY AND fbGetTime.ERR  THEN
			iStateZeit:=0;
		END_IF
	END_CASE

// Auswertung Timetable
	bValueChanged:=FALSE;
	IF tLDate.wMinute <> wLastMinute THEN
		IF 		(arrTimeControl[iRow].wDayOfWeek 	=tLDate.wDayOfWeek+1  
				OR arrTimeControl[iRow].wDayOfWeek = 8 
				OR (arrTimeControl[iRow].wDayOfWeek = 9 AND (tLDate.wDayOfWeek = 0 OR tLDate.wDayOfWeek = 6))
				OR (arrTimeControl[iRow].wDayOfWeek = 10 AND tLDate.wDayOfWeek >=1 AND tLDate.wDayOfWeek <=5))
			AND arrTimeControl[iRow].wHour		=tLDate.wHour
			AND arrTimeControl[iRow].wMinute		=tLDate.wMinute THEN
			nOutputValue:=arrTimeControl[iRow].nValue;
			bValueChanged:=TRUE;
			iRow:=0;
			wLastMinute:=tLDate.wMinute;	
		ELSIF arrTimeControl[iRow].wDayOfWeek = 99 THEN
			iRow:=0;
			wLastMinute:=tLDate.wMinute;
			//nOutputValue:=nInputValue;
		ELSE
			iRow:=iRow+1;
			IF iRow = 50 THEN
				iRow:=0;
				wLastMinute:=tLDate.wMinute;
				//nOutputValue:=nInputValue;
			END_IF
		END_IF
	END_IF

// Abspeichern des Arrays
IF bSafe_Table THEN 
	CASE iState_safe OF
		0:	// Datei anlegen
			iRow_safe:=0;
			fbFileOpen(
				bExecute:=FALSE,
				);
			
			fbFileOpen(
				sNetID:='',
				sPathName:=sFilePath,
				nMode:=FOPEN_MODEAPPEND,
				//ePath:=ePath,
				bExecute:=TRUE,
				tTimeout:=T#5S,
				);
			iState_safe:=iState_safe+1;
			
		1:	// warten bis Funktionsbaustein fertig
			fbFileOpen(
				bExecute:=FALSE,
				);
			IF NOT fbFileOpen.bBusy THEN
				IF fbFileOpen.bError THEN
					iFileOpen_errID:=fbFileOpen.nErrId;
					iState_safe:=0;
				ELSE
					hFile:=fbFileOpen.hFile;
					iFileOpen_errID:=fbFileOpen.nErrId;
					iState_safe:=10;
				END_IF	
			END_IF
			
		
		10:	// Tabellenzeile vorbereiten
			(*fbFormatString(
				sFormat	:= '%S%S%S%S%S%S%S',
				arg1	:= F_STRING(WORD_TO_STRING(arrTimeControl[iRow_safe].wDayOfWeek)),
				arg2	:= F_STRING(sDelimiter),
				arg3	:= F_STRING(WORD_TO_STRING(arrTimeControl[iRow_safe].wHour)),
				arg4	:= F_STRING(sDelimiter),
				arg5	:= F_STRING(WORD_TO_STRING(arrTimeControl[iRow_safe].wMinute)),
				arg6	:= F_STRING(sDelimiter),
				arg7	:= F_STRING(LREAL_TO_STRING(arrTimeControl[iRow_safe].nValue)),
				sOut	=> sString,
				bError	=> bFormatString_error,
				nErrId	=> nFormatString_errID
				);*)
				
		sString:=CONCAT(WORD_TO_STRING(tLDate.wYear),'-');
		IF tLDate.wMonth < 10 THEN
			sString:=CONCAT(sString,'0');
		END_IF
		sString:=CONCAT(sString,WORD_TO_STRING(tLDate.wMonth));
		sString:=CONCAT(sString,'-');
		IF tLDate.wDay < 10 THEN
			sString:=CONCAT(sString,'0');
		END_IF
		sString:=CONCAT(sString,WORD_TO_STRING(tLDate.wDay));
		sString:=CONCAT(sString,sDelimiter);
		sString:=CONCAT(sString,WORD_TO_STRING(tLDate.wHour));
		sString:=CONCAT(sString,':');
		IF tLDate.wMinute < 10 THEN
			sString:=CONCAT(sString,'0');
		END_IF
		sString:=CONCAT(sString,WORD_TO_STRING(tLDate.wMinute));
		sString:=CONCAT(sString,sSpaces);
		sString:=CONCAT(sString,'Uhr');
		sString:=CONCAT(sString,'$09$0A');
		iState_safe:=12;
		
		11:
		sString:=CONCAT(WORD_TO_STRING(arrTimeControl[iRow_safe].wDayOfWeek),sDelimiter);
		sString:=CONCAT(sString,WORD_TO_STRING(arrTimeControl[iRow_safe].wHour));
		sString:=CONCAT(sString,sDelimiter);
		sString:=CONCAT(sString,WORD_TO_STRING(arrTimeControl[iRow_safe].wMinute));
		sString:=CONCAT(sString,sDelimiter);
		sString:=CONCAT(sString,LREAL_TO_STRING(arrTimeControl[iRow_safe].nValue));
		sString:=CONCAT(sString,'$09$0A');
		iRow_safe:=iRow_safe+1;
		iState_safe:=12;		
	(*	// String für CSV vorbereiten
		fb_CSVbuffer(
			eCmd:=eCmd,
			putValue:=sMeasString_temp,
			pValue:=0,
			cbValue:=0,
			bCRLF:=bCRLF,
			pBuffer:=ADR(sMeasString),
			cbBuffer:=SIZEOF(sMeasString),
			cbSize=>iSize_buffer
			);
		
		sMeasString_temp:='';	
			
		// Zeilenende hinzufügen
		MEMSET(ADR(sMeasString)+iSize_buffer-2,9,1);
		sMeasString:=REPLACE(sMeasString,'$0A',2,FIND(sMeasString,'$09$0A'));

*)
		12:	// Tabelle schreiben
		fbFilePuts(
			sNetID:='',
			hfile:=hFile,
			sLine:=sString,
			bExecute:=TRUE,
			bBusy=>bPuts_busy,
			bError=>bPuts_error,
			nErrId=>iPuts_errorID
			);
			
		// wenn Funktionsbaustein fertig, zum nächsten Datenpunkt springen			
		IF NOT bPuts_busy OR bPuts_error THEN
			fbFilePuts(
				bExecute:=FALSE,
				bBusy=>bPuts_busy,
				bError=>bPuts_error,
				nErrId=>iPuts_errorID
				);
				
			IF bPuts_error THEN
				nError_LogError:=nError_LogError+1;
			END_IF
				
			MEMSET(ADR(sString),0,255);
			IF arrTimeControl[iRow_safe].wDayOfWeek=99 OR iRow_safe = 50  THEN
				iState_safe:=20;
			ELSE
				iState_safe:=11;
			END_IF
		END_IF
		
		20: // Datei schließen
			fbFileClose(
				bExecute:=FALSE,
				);
			fbFileClose(
				sNetId:='',
				hFile:=hFile,
				bExecute:=TRUE,
				tTimeout:=,
				);
			iState_safe:=iState_safe+1;
			
		21: // warten bis Baustein fertig ist
			fbFileClose(
				bExecute:=FALSE,
				);
			IF NOT fbFileClose.bBusy THEN		
				IF fbFileClose.bError THEN
					iFileClose_errID:=fbFileClose.nErrId;
				END_IF
					iFileClose_errID:=fbFileClose.nErrId;
					iState_safe:=30;
			END_IF
			
		30: // Speichervorgang abgschlossen
			bSafe_Table:=FALSE;
			iState_safe:=0;
	END_CASE
END_IF

END_FUNCTION_BLOCK
